// TwinCAT 3 PLC project RT1
// ProgramVersion: 3.1.4026.16
// libraries:
//   Tc2_Standard, * (Beckhoff Automation GmbH)
//   Tc2_System, * (Beckhoff Automation GmbH)
//   Tc2_Utilities, * (Beckhoff Automation GmbH)
//   Tc3_Module, * (Beckhoff Automation GmbH)
//   VisuDialogs, * (System)
// project tree:
//   DUTs/ ST_BasicStats.TcDUT
//   DUTs/Time/ E_WeekDay.TcDUT, stTimeToSchedule2.TcDUT, stTimeToSchedule3.TcDUT
//   / GlobalTextList.TcGTLO, PlcTask.TcTTO, Visualization Manager.TcVMO (not stored)
//   GVLs/ GVL_Const.TcGVL, GVL_TimeMeter.TcGVL, GVL_TimeSch.TcGVL
//   POUs/FBs/ FB_BasicStatistics.TcPOU, FB_HourMeter.TcPOU, FB_LastTimesStats.TcPOU, FB_TimeHandler.TcPOU, FB_BasicTimeScheduler.TcPOU, FB_UpdateTime.TcPOU
//   POUs/FUNs/ F_CmpTimeSchedule.TcPOU, F_CmpTimeStruct.TcPOU, F_DT_ToString.TcPOU
//   POUs/ MAIN.TcPOU, prgTimeHandler.TcPOU, prgTimeStatistics.TcPOU
//   VISUs/ EstatisticaTempo.TcVIS, FuncoesExtras.TcVIS, Hora.TcVIS, Data.TcVIS, ImagePool.TcIPO (not stored), Visualization.TcVIS, ProgramacaoHoraria.TcVIS
// real-time tasks:
//   TASK PlcTask: cycle T#10ms, priority 20, ADS port 351
//   TASK VISU_TASK: cycle T#200000us, priority 30, ADS port 350

CONFIGURATION RT1
    RESOURCE PLC ON TwinCAT3
        TASK PlcTask(INTERVAL := T#10ms, PRIORITY := 20);
        PROGRAM MAIN WITH PlcTask : MAIN;
    END_RESOURCE
END_CONFIGURATION

// ---- DUTs/ST_BasicStats.TcDUT
TYPE ST_BasicStats :
STRUCT
	minimum:LREAL;				//The mimimum of the distribution
	maximum:LREAL;              //The maximum of the distribution
	avg:LREAL;                  //The Average of the distribution
	variance:LREAL;             //The Variance
	standardDeviation:LREAL;    //Standard deviation
END_STRUCT
END_TYPE

// ---- DUTs/Time/E_WeekDay.TcDUT
TYPE E_WeekDay :
	(domingo:=0,
	segunda:=1,
	terca:=2,
	quarta:=3,
	quinta:=4,
	sexta:=5,
	sabado:=6);
END_TYPE

// ---- DUTs/Time/stTimeToSchedule2.TcDUT
TYPE stTimeToSchedule2 :
STRUCT
(*relacao do horario que a programacao horaria e ativa/desativada*)
	bIgnore:BOOL;		(*Relevante para desligar TRUE==>> nao desligar*)
	wHour:WORD;			(*Hora exata em que a saida sera acionada/desacionada*)
	wMinute:WORD;		(*Minuto exato em que a saida sera acionada/desacionada*)
	wSecond:WORD;		(*Segundo exato em que a saida sera acionada/desacionada*)
END_STRUCT
END_TYPE

// ---- DUTs/Time/stTimeToSchedule3.TcDUT
TYPE stTimeToSchedule3 :
STRUCT
	bUse:BOOL;			(*Relevante para desligar TRUE==>> nao desligar*)
	wHour:WORD;			(*Hora exata em que a saida sera acionada/desacionada*)
	wMinute:WORD;		(*Minuto exato em que a saida sera acionada/desacionada*)
	wSecond:WORD;		(*Segundo exato em que a saida sera acionada/desacionada*)	
END_STRUCT
END_TYPE

// ---- GVLs/GVL_Const.TcGVL
{attribute 'qualified_only'}
VAR_GLOBAL CONSTANT
	lastStatsValue:UDINT:=10;
END_VAR

// ---- GVLs/GVL_TimeMeter.TcGVL
{attribute 'qualified_only'}
VAR_GLOBAL
	enableTimeCount: BOOL;
	resetTimeCount: BOOL;
	currTaskTime:LREAL;
END_VAR
VAR_GLOBAL PERSISTENT
	hourCounting:LREAL;//
END_VAR

// ---- GVLs/GVL_TimeSch.TcGVL
{attribute 'qualified_only'}
VAR_GLOBAL CONSTANT
	cNumberOfEventSchedules:UINT:=8;//Quantidade de eventos necessarios/programados
(*Não alterar os valores daqui em diante*)
	ciSunday:WORD:=0;				//domingo
	ciMonday:WORD:=1;				//segunda
	ciTuesday:WORD:=2;				//terça
	ciWednesday:WORD:=3;			//quarta
	ciThursday:WORD:=4;				//quinta
	ciFriday:WORD:=5;				//sexta
	ciSaturday:WORD:=6;				//sabado
END_VAR
VAR_GLOBAL
	//Data e hora atuais
	actualDate:TIMESTRUCT;				//Data/Hora autais
	sActualDate: STRING;				(*String com a data atual*)
	sActualTime: STRING;				(*String com a hora atual*)
	sWeekDay:STRING;					(*Dia da semana*)
	//Acertar a hora
	timeToInsert: TIMESTRUCT;			//Hora a inserir (acertar hora)
	bUpdateTime: BOOL;					(*Atualizar a hora*)
	bUpdateDate: BOOL;					(*Atualizar a data*)
	(*Estrutura contendo a data e hora a serem inseridas*)	
	//Variaveis especificas da programacao horaria
	abOutScheduler:ARRAY[1..cNumberOfEventSchedules] OF BOOL;//Variaveis ativadas pelo bloco de programacao horaria
	uiIndexToCheck:UINT:=1;									//Index
	abErr:ARRAY[1..cNumberOfEventSchedules] OF BOOL;		//Erro na programacao horaria
	asErr:ARRAY[1..cNumberOfEventSchedules] OF STRING;		//
	bTurnOffOutput: BOOL;									//Desliga a saida dos blocos de 
END_VAR
VAR_GLOBAL PERSISTENT
	aTimeToSchActivate:ARRAY[0..6,1..cNumberOfEventSchedules] OF stTimeToSchedule3;		//Hora de ativar
	aTimeToSchDeactivate:ARRAY[0..6,1..cNumberOfEventSchedules] OF stTimeToSchedule3;	//Hora de desativar
END_VAR
//GVL_TimeSchBABR

// ---- POUs/MAIN.TcPOU
PROGRAM MAIN
VAR

END_VAR

prgTimeHandler();

prgTimeStatistics();

END_PROGRAM

// ---- POUs/prgTimeHandler.TcPOU
(*
	Programa realiza o gerenciamento da programacao horaria
	Esta rotina deve ser chamada no "MAIN" 
*)
PROGRAM prgTimeHandler
VAR
	timeScheduler:ARRAY[1..GVL_TimeSch.cNumberOfEventSchedules] OF FB_BasicTimeScheduler;
	i: UINT;
	timer:FB_TimeHandler;				(*Obtem a hora do sistema*)
	updateTime:FB_UpdateTime;			(*Bloco *)
	sActualTime: STRING;
	dt1: DATE_AND_TIME;
	timeMeter:FB_HourMeter;
	taskInfo: PlcTaskSystemInfo;
	bError: BOOL;
	sErr: STRING;
END_VAR

(*Le a data / Hora do sistema*)
timer(
	bDisplaySecond:= TRUE, 
	bShowDateNumberFormat:= TRUE, 
	sWeekDay=> GVL_TimeSch.sWeekDay, 
	sActualTime=> GVL_TimeSch.sActualTime, 
	sActualDate=> GVL_TimeSch.sActualDate, 
	outStruct=> GVL_TimeSch.actualDate);

(*Responsavel por atualizar a data/hora do sistema*)
updateTime(
	timeToInsert:= GVL_TimeSch.timeToInsert ,
	actualTime:= GVL_TimeSch.actualDate,
	bUpdateTime:= GVL_TimeSch.bUpdateTime,
	bUpdateDate:= GVL_TimeSch.bUpdateDate,
	bError=> ,
	iErrorId=> );

(*blocos de programacao horaria*)
FOR i := 1 TO GVL_TimeSch.cNumberOfEventSchedules DO
	timeScheduler[i](
		timeToActivate:= GVL_TimeSch.aTimeToSchActivate[GVL_TimeSch.actualDate.wDayOfWeek,i], 
		timeToDeactivate:= GVL_TimeSch.aTimeToSchDeactivate[GVL_TimeSch.actualDate.wDayOfWeek,i], 
		actualTime:= GVL_TimeSch.actualDate,
		bTurnOffOutput:= GVL_TimeSch.bTurnOffOutput,
		bErr=> GVL_TimeSch.abErr[i],
		sErr=> GVL_TimeSch.asErr[i],
		bOut=> GVL_TimeSch.abOutScheduler[i]);
END_FOR


taskInfo:=_TaskInfo[1];

sActualTime:=F_DT_ToString(dt1);

GVL_TimeMeter.currTaskTime:= UDINT_TO_LREAL(taskInfo.CycleTime)/10E6;

timeMeter(
	enableCount:= GVL_TimeMeter.enableTimeCount, 
	resetCount:= GVL_TimeMeter.resetTimeCount, 
	cycleTime:= GVL_TimeMeter.currTaskTime, 
	bError=>bError, 
	sErr=> sErr, 
	pastTime:=GVL_TimeMeter.hourCounting );

END_PROGRAM

// ---- POUs/FBs/FB_BasicTimeScheduler.TcPOU
FUNCTION_BLOCK FB_BasicTimeScheduler
VAR_INPUT
	timeToActivate:stTimeToSchedule3;		//Hora para ativar a saída
	timeToDeactivate:stTimeToSchedule3;		//Hora para desativar a saída
	actualTime:TIMESTRUCT;					//Hora/Data atual
	bTurnOffOutput:BOOL;					//Desliga a saída imediatamente
END_VAR
VAR_OUTPUT
	bErr: BOOL;
	sErr:STRING;
	bOut:BOOL;
END_VAR
VAR
	timeToActivateR_TRIG:R_TRIG;
	timeToDeactivateR_TRIG:R_TRIG;
END_VAR

sErr:='';
bErr:=FALSE;
IF NOT M_CheckTimeSchedule(timeToActivate) OR NOT (M_CheckTimeSchedule(timeToDeactivate) OR NOT timeToDeactivate.bUse) THEN
	bErr:=TRUE;
	sErr:='Parâmetros invalidos';
END_IF

timeToActivateR_TRIG(CLK:= M_CmpTimeStr_Schedule(actualTime,timeToActivate));
timeToDeactivateR_TRIG(CLK:= M_CmpTimeStr_Schedule(actualTime,timeToDeactivate));

IF timeToActivateR_TRIG.Q AND NOT bTurnOffOutput AND NOT bErr AND timeToActivate.bUse THEN
	bOut:=TRUE;
END_IF
IF timeToDeactivateR_TRIG.Q AND timeToDeactivate.bUse THEN
	bOut:=FALSE;
END_IF
IF bTurnOffOutput THEN
	bOut:=FALSE;
END_IF

METHOD M_CheckTimeSchedule : BOOL
VAR_INPUT
	timeSchedule:stTimeToSchedule3;	//Hora marcada a ser validada
END_VAR
M_CheckTimeSchedule:= (timeSchedule.wHour>=0 AND timeSchedule.wHour<=23)AND (timeSchedule.wMinute>=0 AND timeSchedule.wMinute <=59)
AND (timeSchedule.wSecond>=0 AND timeSchedule.wSecond <=59);
END_METHOD

METHOD PRIVATE M_CmpTimeStr_Schedule : BOOL
VAR_INPUT
	actualTime:TIMESTRUCT;
	scheduledTime:stTimeToSchedule3;
END_VAR
VAR
	timeToCmp:TIMESTRUCT;
END_VAR
(*
	Esse metodo retorna true caso a hora atual seja >= à hora marcada para ocorrer o evento
	Caso a variave 'bUse' do tempo marcado esteja desabilita também retorna false
*)
timeToCmp.wYear:=actualTime.wYear;
timeToCmp.wMonth:=actualTime.wMonth;
timeToCmp.wDay:=actualTime.wDay;
timeToCmp.wDayOfWeek:=actualTime.wDayOfWeek;
timeToCmp.wHour:=scheduledTime.wHour;
timeToCmp.wMinute:= scheduledTime.wMinute;
timeToCmp.wSecond:=scheduledTime.wSecond;
M_CmpTimeStr_Schedule:=F_CmpTimeStruct(actualTime,timeToCmp);
END_METHOD

END_FUNCTION_BLOCK

// ---- POUs/FUNs/F_CmpTimeStruct.TcPOU
FUNCTION F_CmpTimeStruct : BOOL
VAR_INPUT
	time1:TIMESTRUCT;
	time2:TIMESTRUCT;
END_VAR
VAR
END_VAR
(*Esta funcao verifica se a TimeStruct fornecida é válida
a variavel "time1"devera ser maior que a  variavel "time2" para que a funcao seja verdadeira*)

F_CmpTimeStruct:= SYSTEMTIME_TO_DT( time1)>SYSTEMTIME_TO_DT( time2);

END_FUNCTION

// ---- POUs/FBs/FB_TimeHandler.TcPOU
FUNCTION_BLOCK FB_TimeHandler
VAR_INPUT
	bDisplaySecond:BOOL;			(*Mostra os segundos na variavel de saida de hora*)
	bShowDateNumberFormat:BOOL;	(*Mostra a data em formato numerico (e.g.: 01/01/1970)*)
END_VAR
VAR_OUTPUT
	sActualMonth: STRING;			(*Mes do ano*)
	sWeekDay:STRING;				(*Dia da semana*)
	sActualTime:STRING;				(*Hora*)
	sActualDate:STRING;				(*Data atual*)
	outStruct:TIMESTRUCT;
END_VAR
VAR
	getTime:FB_LocalSystemTime;		(*Obtem a data/hora do sistema*)
	sSecond: STRING;
END_VAR


(*Obtem a hora do Windows*)
getTime(
	sNetID:='' ,
	bEnable:=TRUE ,
	dwCycle:= ,
	dwOpt:= ,
	tTimeout:= ,
	bValid=> ,
	tzID=> );

ASetStrings();
outStruct:=getTime.systemTime;

ACTION ASetStrings:
IF getTime.bValid THEN
	CASE getTime.systemTime.wMonth OF
		1:
			sActualMonth:='Janeiro';
		2:
			sActualMonth:='Fevereiro';
		3:
			sActualMonth:='Março';
		4:
			sActualMonth:='Abril';
		5:
			sActualMonth:='Maio';
		6:
			sActualMonth:='Junho';
		7:
			sActualMonth:='Julho';
		8:
			sActualMonth:='Agosto';
		9:
			sActualMonth:='Setembro';
		10:
			sActualMonth:='Outubro';
		11:
			sActualMonth:='Novembro';
		12:
			sActualMonth:='Dezembro';
	END_CASE

	CASE getTime.systemTime.wDayOfWeek OF
		0:
			sWeekDay:='Domingo';
		1:
			sWeekDay:='Segunda';
		2:
			sWeekDay:='Terça';
		3:
			sWeekDay:='Quarta';
		4:
			sWeekDay:='Quinta';
		5:
			sWeekDay:='Sexta';
		6:
			sWeekDay:='Sabado';
	END_CASE
	sSecond:=SEL(getTime.systemTime.wSecond<10,WORD_TO_STRING(getTime.systemTime.wSecond),CONCAT('0',WORD_TO_STRING(getTime.systemTime.wSecond)));

	sActualTime:=CONCAT(WORD_TO_STRING(getTime.systemTime.wHour),CONCAT(':',CONCAT(WORD_TO_STRING(getTime.systemTime.wMinute),SEL(bDisplaySecond,'',CONCAT(':',sSecond)))));

	IF NOT bShowDateNumberFormat THEN
		sActualDate:=CONCAT(WORD_TO_STRING(getTime.systemTime.wDay),CONCAT(' de ',CONCAT(sActualMonth,CONCAT(' de ' ,WORD_TO_STRING(getTime.systemTime.wYear)))));
	ELSE
		sActualDate:=CONCAT(WORD_TO_STRING(getTime.systemTime.wDay),CONCAT('/',CONCAT(WORD_TO_STRING(getTime.systemTime.wMonth),CONCAT('/',WORD_TO_STRING(getTime.systemTime.wYear)))));
	END_IF
ELSE
	sActualDate:='????';
	sActualTime:='????';
	sWeekDay:='????';
	sActualMonth:='????';
END_IF
END_ACTION

END_FUNCTION_BLOCK

// ---- POUs/FBs/FB_UpdateTime.TcPOU
FUNCTION_BLOCK FB_UpdateTime
VAR_INPUT
	timeToInsert:TIMESTRUCT;		(*estruta com data/hora a ser inserida*)
	actualTime:TIMESTRUCT;			(*estrutura contendo a data/hora atual*)
	bUpdateTime: BOOL;				(*atualiza a hora com um pulso nessa entrada*)
	bUpdateDate: BOOL;				(*atualiza a data com um pulso nessa entrada*)
END_VAR
VAR_OUTPUT
	bError: BOOL;						(*Erro ativo*)
	iErrorId: UDINT;					(*Id do erro*)
END_VAR
VAR
	setTime:NT_SetLocalTime;			(*Funcao para atualizar a data/hora*)
END_VAR

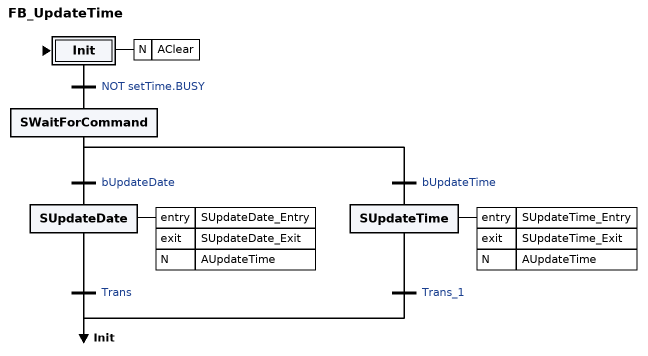
INITIAL_STEP Init:
    AClear(N);
END_STEP
TRANSITION FROM Init TO SWaitForCommand
    := NOT setTime.BUSY;
END_TRANSITION
STEP SWaitForCommand:
END_STEP
TRANSITION FROM SWaitForCommand TO SUpdateDate
    := bUpdateDate;
END_TRANSITION
STEP SUpdateDate:
    SUpdateDate_Entry(P1);  // entry action
    SUpdateDate_Exit(P0);  // exit action
    AUpdateTime(N);
END_STEP
TRANSITION FROM SUpdateDate TO Init
    := Trans;
END_TRANSITION
TRANSITION FROM SWaitForCommand TO SUpdateTime
    := bUpdateTime;
END_TRANSITION
STEP SUpdateTime:
    SUpdateTime_Entry(P1);  // entry action
    SUpdateTime_Exit(P0);  // exit action
    AUpdateTime(N);
END_STEP
TRANSITION FROM SUpdateTime TO Init
    := Trans_1;
END_TRANSITION

ACTION AClear:
setTime(	NETID:='' ,START:=FALSE );
END_ACTION

ACTION AUpdateTime:
setTime(
	NETID:='' ,
	START:= TRUE,
	ERR=>bError ,
	ERRID=> iErrorId);
END_ACTION

ACTION SUpdateDate_Entry:
(*Inicia o processo de atualizar a data*)


setTime.TIMESTR:=actualTime;
setTime.TIMESTR.wDay:=timeToInsert.wDay;
setTime.TIMESTR.wMonth:=timeToInsert.wMonth;
setTime.TIMESTR.wYear:=timeToInsert.wYear;
END_ACTION

ACTION SUpdateDate_Exit:
setTime(	NETID:='' ,START:=FALSE );
END_ACTION

ACTION SUpdateTime_Entry:
(*Inicia o processo de atualizar a data*)


setTime.TIMESTR:=actualTime;

setTime.TIMESTR.wHour:=timeToInsert.wHour;
setTime.TIMESTR.wMinute:=timeToInsert.wMinute;
setTime.TIMESTR.wSecond:=timeToInsert.wSecond;
END_ACTION

ACTION SUpdateTime_Exit:
setTime(	NETID:='' ,START:=FALSE );
END_ACTION

TRANSITION Trans:
NOT setTime.BUSY
END_TRANSITION

TRANSITION Trans_1:
NOT setTime.BUSY
END_TRANSITION

END_FUNCTION_BLOCK

// ---- POUs/FBs/FB_HourMeter.TcPOU
FUNCTION_BLOCK FB_HourMeter
VAR_INPUT
	enableCount: BOOL;	//this variable enables the time count
	resetCount:BOOL;	//set it to true in order to reset the whole count
	cycleTime:LREAL;	//cycle time in seconds
END_VAR
VAR_OUTPUT
	bError:BOOL;
	sErr:STRING;
END_VAR
VAR_IN_OUT
	pastTime:LREAL;	//Variable that contains the time past, should be persistent/retain outside the block otherwise the time count will not 
					//be kept once the PLC is stopped
END_VAR
VAR
	m:BOOL;			//memory to activate the rising trigger to reset the counter
END_VAR

IF enableCount AND cycleTime>0.0 THEN
	pastTime:= pastTime + cycleTime/3600;
	bError:=FALSE;
	sErr:='';
ELSIF cycleTime <=0 THEN
	bError:=TRUE;
	sErr:= 'wrong configured time';
END_IF


IF resetCount AND NOT m THEN
	pastTime:=0;
END_IF
m := resetCount;

END_FUNCTION_BLOCK

// ---- POUs/FUNs/F_DT_ToString.TcPOU
FUNCTION F_DT_ToString : STRING
VAR_INPUT
	in:DATE_AND_TIME;
END_VAR
VAR
	tsDtToConvert:TIMESTRUCT;
END_VAR

tsDtToConvert:= DT_TO_SYSTEMTIME(in);

F_DT_ToString:= CONCAT(WORD_TO_STRING(tsDtToConvert.wDay),'/');
F_DT_ToString:= CONCAT(F_DT_ToString, CONCAT( WORD_TO_STRING(tsDtToConvert.wMonth),'/'));
F_DT_ToString:= CONCAT(F_DT_ToString, CONCAT( WORD_TO_STRING(tsDtToConvert.wYear),'/'));
F_DT_ToString:= CONCAT(F_DT_ToString, ' ');
F_DT_ToString:= CONCAT(F_DT_ToString, CONCAT( WORD_TO_STRING(tsDtToConvert.wHour),':'));
F_DT_ToString:= CONCAT(F_DT_ToString, CONCAT( WORD_TO_STRING(tsDtToConvert.wMinute),':'));
F_DT_ToString:= CONCAT(F_DT_ToString,  WORD_TO_STRING(tsDtToConvert.wSecond));

END_FUNCTION

// ---- POUs/prgTimeStatistics.TcPOU
PROGRAM prgTimeStatistics
VAR
	enableTimeCount: BOOL;
	lastTimeStats:FB_LastTimesStats;
	stats:st_BasicStats;
	lastTime: TIME;
	currTime: TIME;
	lastTimes: ARRAY [1..GVL_Const.lastStatsValue] OF TIME;
	arLastTimes: ARRAY [1..GVL_Const.lastStatsValue] OF LREAL;
END_VAR

lastTimeStats(enable:= enableTimeCount,lastTime => lastTime, currTime=>currTime, lastTimes => lastTimes, arLastTimes => arLastTimes);

stats:=lastTimeStats.M_GetBasicStats();

END_PROGRAM

// ---- POUs/FBs/FB_LastTimesStats.TcPOU
FUNCTION_BLOCK FB_LastTimesStats EXTENDS FB_BasicStatistics
VAR_INPUT
	enable: BOOL;	//Enable time counting
END_VAR
VAR_OUTPUT
	lastTime:TIME;
	currTime:TIME;
	lastTimes:ARRAY[1..GVL_Const.lastStatsValue] OF TIME;
	arLastTimes:ARRAY[1..GVL_Const.lastStatsValue] OF LREAL;
END_VAR
VAR
	t1:TON;
	disableTrig:F_TRIG;
	i: UDINT;
END_VAR

disableTrig(CLK:= enable);
IF disableTrig.Q THEN
	lastTime:= t1.ET;
	FOR i:= GVL_Const.lastStatsValue TO 2 BY -1 DO
		lastTimes[i]:= lastTimes[i-1];
	END_FOR
	lastTimes[1]:=lastTime;
	FOR i:= 1 TO GVL_Const.lastStatsValue DO
		arLastTimes[i]:= TIME_TO_LREAL(lastTimes[i])/1000;
	END_FOR
END_IF
t1(IN:= enable, PT:= T#7D);
currTime:= t1.ET;

METHOD M_GetBasicStats : ST_BasicStats
VAR_INPUT
END_VAR
M_GetBasicStats.avg:=SUPER^.M_CalcAvg(THIS^.arLastTimes);
M_GetBasicStats.maximum:=SUPER^.M_CalcMax(THIS^.arLastTimes);
M_GetBasicStats.minimum:=SUPER^.M_CalcMin(THIS^.arLastTimes);
M_GetBasicStats.variance:=SUPER^.M_CalcVariance(THIS^.arLastTimes);
M_GetBasicStats.standardDeviation:=SUPER^.M_CalcSD(THIS^.arLastTimes);
END_METHOD

END_FUNCTION_BLOCK

// ---- POUs/FBs/FB_BasicStatistics.TcPOU
FUNCTION_BLOCK FB_BasicStatistics
VAR_INPUT
END_VAR
VAR_OUTPUT
END_VAR
VAR
END_VAR

METHOD M_CalcAvg : LREAL
VAR_IN_OUT
	valuesToAvg:ARRAY[*] OF LREAL;
END_VAR
VAR
	i: DINT;
	sum:LREAL;
	numOfElements: LREAL;
END_VAR
sum:=0;
numOfElements:=0;
FOR i := LOWER_BOUND(valuesToAvg,1) TO UPPER_BOUND(valuesToAvg,1) DO
	sum:= sum+ valuesToAvg[i];
	numOfElements:=numOfElements+1;
END_FOR
IF numOfElements >0 THEN
	M_CalcAvg :=sum/numOfElements;
END_IF
END_METHOD

METHOD M_CalcMax : LREAL
VAR_IN_OUT
	valuesToMax:ARRAY[*] OF LREAL;
END_VAR

VAR
	maximum: LREAL;
	i: DINT;
END_VAR
maximum:=valuesToMax[1];
FOR i:= LOWER_BOUND(valuesToMax,1) TO UPPER_BOUND(valuesToMax,1) DO
	maximum:= MAX(maximum,valuesToMax[i]);
END_FOR
M_CalcMax:= maximum;
END_METHOD

METHOD M_CalcMin : LREAL
VAR_IN_OUT
	valuesToMin:ARRAY[*] OF LREAL;
END_VAR

VAR
	minimum: LREAL;
	i: DINT;
END_VAR
minimum:=valuesToMin[1];
FOR i:= LOWER_BOUND(valuesToMin,1) TO UPPER_BOUND(valuesToMin,1) DO
	minimum:= MIN(minimum,valuesToMin[i]);
END_FOR
M_CalcMin:= minimum;
END_METHOD

METHOD M_CalcSD : LREAL
VAR_INPUT
	valuesToSD:ARRAY[1..GVL_Const.lastStatsValue] OF LREAL;
END_VAR
M_CalcSD := SQRT(M_CalcVariance(valuesToSD));
END_METHOD

METHOD PUBLIC M_CalcVariance : LREAL
VAR_IN_OUT
	valuesToVar:ARRAY[*] OF LREAL;
END_VAR
VAR
	i: DINT;
	sum:LREAL;
	avg:LREAL;
	numOfElements:lreal;
END_VAR
sum:=numOfElements:=0;
avg:= M_CalcAvg(valuesToVar);
FOR i := LOWER_BOUND(valuesToVar,1) TO UPPER_BOUND(valuesToVar,1) DO
	sum:= sum+EXPT(valuesToVar[i]-avg,2);
	numOfElements:= numOfElements+1;
END_FOR
M_CalcVariance:= sum/numOfElements;
END_METHOD

END_FUNCTION_BLOCK

// ---- POUs/FUNs/F_CmpTimeSchedule.TcPOU
FUNCTION F_CmpTimeSchedule : BOOL
VAR_INPUT
	timeToActivate:stTimeToSchedule2;	(*Hora para ligar a saida*)
	timeToDeactivate:stTimeToSchedule2;	(*Hora para desligar a saida*)
END_VAR
VAR
END_VAR

F_CmpTimeSchedule:=(timeToDeactivate.wHour>timeToActivate.wHour) OR ((timeToDeactivate.wHour = timeToActivate.wHour) AND (timeToDeactivate.wMinute> timeToActivate.wMinute));

END_FUNCTION

// ---- GlobalTextList.TcGTLO
TEXTLIST GlobalTextList
  148 = '%.1f'
  509 = '%d'
  18 = '%s'
  793 = '%t'
  615 = '180'
  9 = 'Acertar Data'
  8 = 'Acertar Hora'
  12 = 'Ano'
  19 = 'Ativar'
  88 = 'Atual'
  7 = 'Atualizar'
  16 = 'Checkbox'
  0 = 'DATA : %s'
  20 = 'Desativar'
  183 = 'Desvio P.'
  14 = 'dia'
  15 = 'Dia'
  28 = 'Dia : %s'
  26 = 'domingo'
  27 = 'Domingo'
  585 = 'Estats tempo'
  694 = 'Extras'
  986 = 'Habilitar'
  4 = 'Hora'
  1 = 'HORA : %s'
  891 = 'Horas : %.1f'
  13 = 'Mes'
  5 = 'Min'
  876 = 'Máximo'
  277 = 'Médio'
  38 = 'Mínimo'
  783 = 'Programação'
  252 = 'Programação horária'
  22 = 'Quarta'
  23 = 'Quinta'
  287 = 'Reset'
  25 = 'Sabado'
  6 = 'Seg'
  17 = 'Segunda'
  24 = 'Sexta'
  610 = 'T. Ciclo %.2f (s)'
  11 = 'Tela 1'
  10 = 'Tela 2'
  21 = 'Terça'
  3 = 'Update Date'
  2 = 'Update Time'
  181 = 'Variância'
  250 = 'Último'
  665 = 'Últimos tempos'
  29 = 'Últimos tempos (Real)'
  583 = 'Últimos tempos (s)'
  391 = 'Últimos tempos (Segundos)'
  880 = 'Últimos tempos (T)'
END_TEXTLIST

// ---- VISUs/EstatisticaTempo.TcVIS
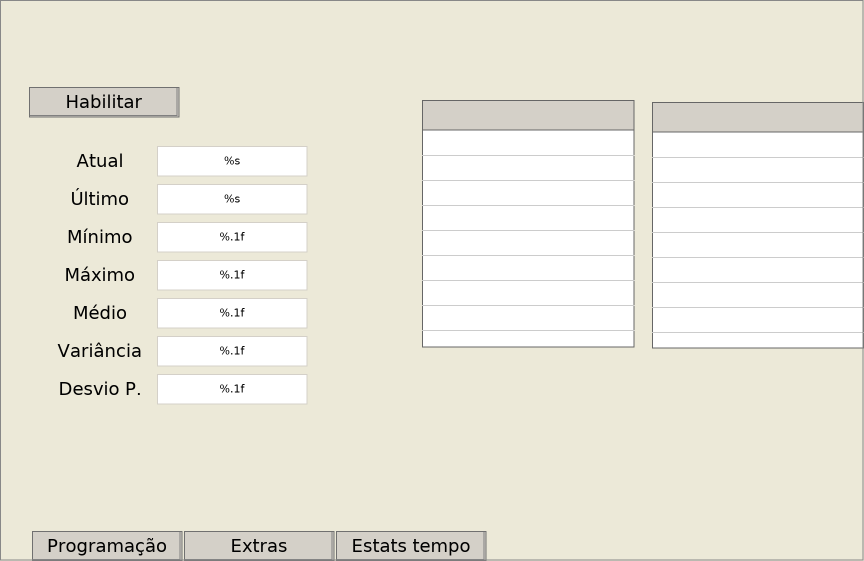
VISUALIZATION EstatisticaTempo  // 864x561
    Button (32,531 150x30), "Programação"
        OnMouseClick: change screen: Visualization
    Button (184,531 150x30), "Extras"
        OnMouseClick: change screen: FuncoesExtras
    Button (336,531 150x30), "Estats tempo"
        OnMouseClick: change screen: EstatisticaTempo
    Table (422,100 212x247), data array: prgTimeStatistics.lastTimes
        p3854506369: prgTimeStatistics.lastTimes[INDEX]
        p2232123230: Últimos tempos (T)
    Table (652,102 212x246), data array: prgTimeStatistics.arLastTimes
        p3854506369: prgTimeStatistics.arLastTimes[INDEX]
        p2232123230: Últimos tempos (s)
    Button (29,87 150x30), "Habilitar"
        toggle prgTimeStatistics.enableTimeCount
    Label (40,146 120x30), "Atual"
    Label (40,184 120x30), "Último"
    Label (40,222 120x30), "Mínimo"
    Label (40,260 120x30), "Máximo"
    Label (40,298 120x30), "Médio"
    Label (40,336 120x30), "Variância"
    Label (40,374 120x30), "Desvio P."
    Textfield (157,146 150x30), "%s", text variable: prgTimeStatistics.lastTimeStats.currTime
    Textfield (157,184 150x30), "%s", text variable: prgTimeStatistics.lastTimeStats.lastTime
    Textfield (157,222 150x30), "%.1f", text variable: prgTimeStatistics.stats.minimum
    Textfield (157,260 150x30), "%.1f", text variable: prgTimeStatistics.stats.maximum
    Textfield (157,298 150x30), "%.1f", text variable: prgTimeStatistics.stats.avg
    Textfield (157,336 150x30), "%.1f", text variable: prgTimeStatistics.stats.variance
    Textfield (157,374 150x30), "%.1f", text variable: prgTimeStatistics.stats.standardDeviation
END_VISUALIZATION

// ---- VISUs/FuncoesExtras.TcVIS
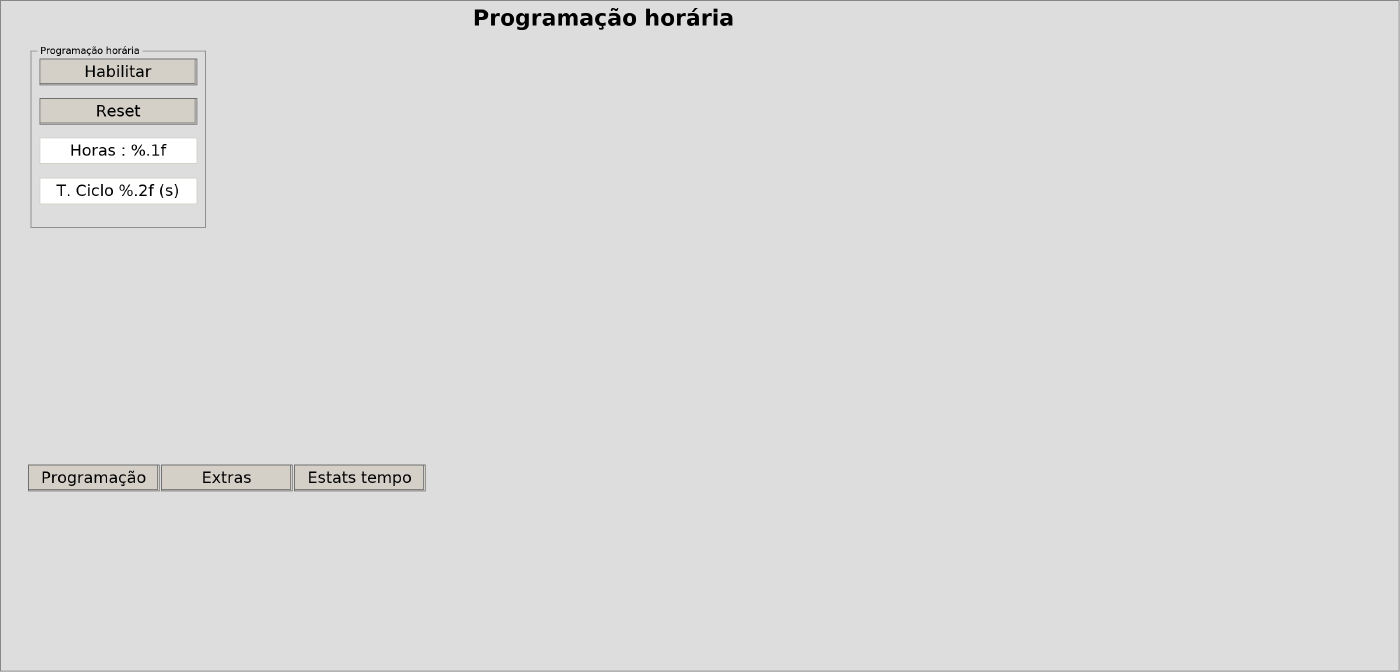
VISUALIZATION FuncoesExtras  // 1600x768
    Label (500,5 380x30), "Programação horária"
    GroupBox (35,50 200x210), "Programação horária"
        Button (10,17 180x30), "Habilitar"
            toggle GVL_TimeMeter.enableTimeCount
        Button (10,62 180x30), "Reset"
            tap GVL_TimeMeter.resetTimeCount
        Textfield (10,107 180x30), "Horas : %.1f", text variable: GVL_TimeMeter.hourCounting
        Textfield (10,153 180x30), "T. Ciclo %.2f (s)", text variable: GVL_TimeMeter.currTaskTime
    Button (32,531 150x30), "Programação"
        OnMouseClick: change screen: Visualization
    Button (184,531 150x30), "Extras"
        OnMouseClick: change screen: FuncoesExtras
    Button (336,531 150x30), "Estats tempo"
        OnMouseClick: change screen: EstatisticaTempo
END_VISUALIZATION

// ---- VISUs/Hora.TcVIS
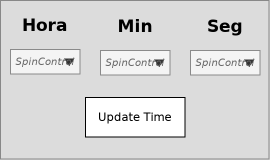
VISUALIZATION Hora  // 270x160
    Rectangle (85,97 100x40), "Update Time"
        tap GVL_TimeSch.bUpdateTime
    SpinControl (10,49 70x25), variable: GVL_TimeSch.timeToInsert.wHour
        OnMouseClick: write the text variable via Default, min 0, max 23
    Label (10,10 70x30), "Hora"
    SpinControl (100,50 70x25), variable: GVL_TimeSch.timeToInsert.wMinute
        OnMouseClick: write the text variable via Default, min 0, max 59
    Label (100,11 70x30), "Min"
    SpinControl (190,50 70x25), variable: GVL_TimeSch.timeToInsert.wSecond
        OnMouseClick: write the text variable via Default, min 0, max 59
    Label (190,11 70x30), "Seg"
END_VISUALIZATION

// ---- VISUs/Data.TcVIS
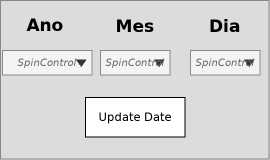
VISUALIZATION Data  // 270x160
    SpinControl (2,50 90x25), variable: GVL_TimeSch.timeToInsert.wYear
        OnMouseClick: write the text variable via Default, min 2000, max 3000
    Label (10,10 70x30), "Ano"
    SpinControl (100,50 70x25), variable: GVL_TimeSch.timeToInsert.wMonth
        OnMouseClick: write the text variable via Default, min 1, max 12
    Label (100,11 70x30), "Mes"
    SpinControl (190,50 70x25), variable: GVL_TimeSch.timeToInsert.wDay
        OnMouseClick: write the text variable via Default, min 1, max 31
    Label (190,11 70x30), "Dia"
    Rectangle (85,97 100x40), "Update Date"
        tap GVL_TimeSch.bUpdateDate
END_VISUALIZATION

// ---- VISUs/Visualization.TcVIS
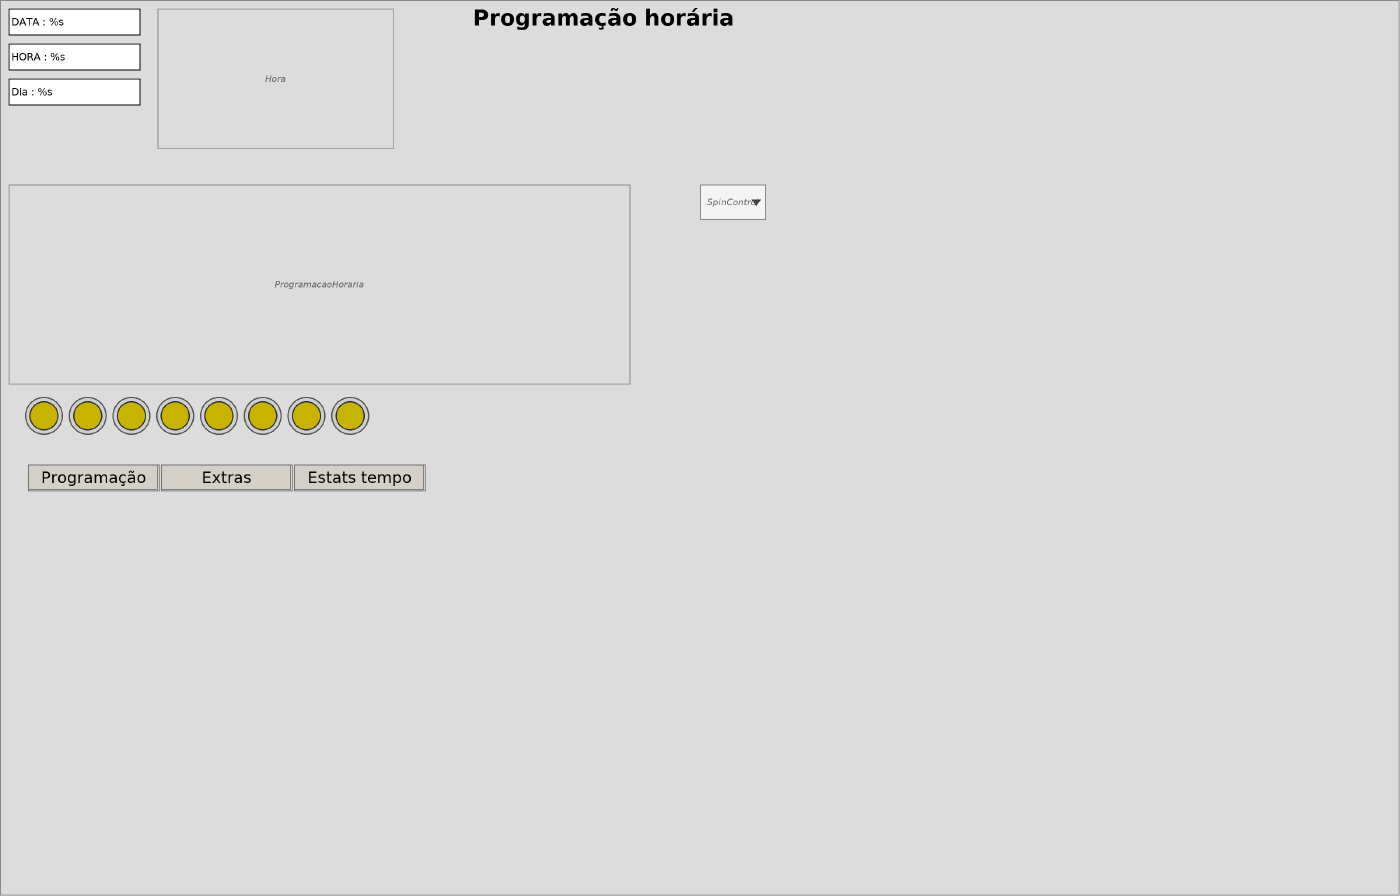
VISUALIZATION Visualization  // 1600x1024
    Rectangle (10,10 150x30), "DATA : %s", text variable: GVL_TimeSch.sActualDate
    Rectangle (10,50 150x30), "HORA : %s", text variable: GVL_TimeSch.sActualTime
    TabControl (180,10 270x160)
        shows Hora()
        shows Data()
        [0]: TabTitle=Acertar Hora
        [1]: TabTitle=Acertar Data
    TabControl (10,211 710x228)
        shows ProgramacaoHoraria(uiIndex := GVL_TimeSch.uiIndexToCheck, wDayOfWeek := GVL_TimeSch.ciMonday)
        shows ProgramacaoHoraria(uiIndex := GVL_TimeSch.uiIndexToCheck, wDayOfWeek := GVL_TimeSch.ciTuesday)
        shows ProgramacaoHoraria(uiIndex := GVL_TimeSch.uiIndexToCheck, wDayOfWeek := GVL_TimeSch.ciWednesday)
        shows ProgramacaoHoraria(uiIndex := GVL_TimeSch.uiIndexToCheck, wDayOfWeek := GVL_TimeSch.ciThursday)
        shows ProgramacaoHoraria(uiIndex := GVL_TimeSch.uiIndexToCheck, wDayOfWeek := GVL_TimeSch.ciFriday)
        shows ProgramacaoHoraria(uiIndex := GVL_TimeSch.uiIndexToCheck, wDayOfWeek := GVL_TimeSch.ciSaturday)
        shows ProgramacaoHoraria(uiIndex := GVL_TimeSch.uiIndexToCheck, wDayOfWeek := GVL_TimeSch.ciSunday)
        [0]: TabTitle=Segunda
        [1]: TabTitle=Terça
        [2]: TabTitle=Quarta
        [3]: TabTitle=Quinta
        [4]: TabTitle=Sexta
        [5]: TabTitle=Sabado
        [6]: TabTitle=Domingo
    Rectangle (10,90 150x30), "Dia : %s", text variable: GVL_TimeSch.sWeekDay
    SpinControl (800,211 75x40), variable: GVL_TimeSch.uiIndexToCheck
        p651134158: GVL_TimeSch.cNumberOfEventSchedules
    Group (25,450 400x50)
        Lamp1 (0,0 50x50), variable: GVL_TimeSch.abOutScheduler[1], style: Lamp-Lamp1-Yellow
        Lamp1 (50,0 50x50), variable: GVL_TimeSch.abOutScheduler[2], style: Lamp-Lamp1-Yellow
        Lamp1 (100,0 50x50), variable: GVL_TimeSch.abOutScheduler[3], style: Lamp-Lamp1-Yellow
        Lamp1 (150,0 50x50), variable: GVL_TimeSch.abOutScheduler[4], style: Lamp-Lamp1-Yellow
        Lamp1 (200,0 50x50), variable: GVL_TimeSch.abOutScheduler[5], style: Lamp-Lamp1-Yellow
        Lamp1 (250,0 50x50), variable: GVL_TimeSch.abOutScheduler[6], style: Lamp-Lamp1-Yellow
        Lamp1 (300,0 50x50), variable: GVL_TimeSch.abOutScheduler[7], style: Lamp-Lamp1-Yellow
        Lamp1 (350,0 50x50), variable: GVL_TimeSch.abOutScheduler[8], style: Lamp-Lamp1-Yellow
    Label (500,5 380x30), "Programação horária"
    Button (32,531 150x30), "Programação"
        OnMouseClick: change screen: Visualization
    Button (184,531 150x30), "Extras"
        OnMouseClick: change screen: FuncoesExtras
    Button (336,531 150x30), "Estats tempo"
        OnMouseClick: change screen: EstatisticaTempo
END_VISUALIZATION

// ---- VISUs/ProgramacaoHoraria.TcVIS
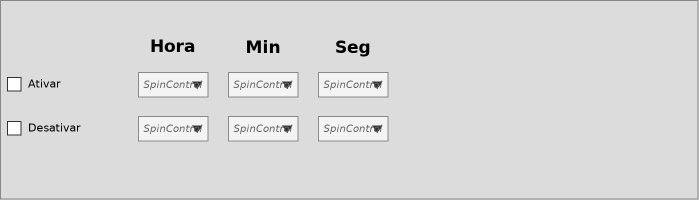
VISUALIZATION ProgramacaoHoraria  // 699x200
VAR_IN_OUT

END_VAR
VAR_INPUT
	uiIndex:UINT;		//Indice da programacao horaria
	wDayOfWeek:WORD;	
END_VAR
    Checkbox (5,69 120x30), "Ativar", variable: GVL_TimeSch.aTimeToSchActivate[wDayOfWeek,uiIndex].bUse
    Checkbox (5,113 120x30), "Desativar", variable: GVL_TimeSch.aTimeToSchDeactivate[wDayOfWeek,uiIndex].bUse
    SpinControl (138,72 70x25), variable: GVL_TimeSch.aTimeToSchActivate[wDayOfWeek,uiIndex].wHour
        OnMouseClick: write the text variable via Default, min 0, max 23
    Label (138,31 70x30), "Hora"
    SpinControl (228,72 70x25), variable: GVL_TimeSch.aTimeToSchActivate[wDayOfWeek,uiIndex].wMinute
        OnMouseClick: write the text variable via Default, min 0, max 59
    Label (228,32 70x30), "Min"
    SpinControl (318,72 70x25), variable: GVL_TimeSch.aTimeToSchActivate[wDayOfWeek,uiIndex].wSecond
        OnMouseClick: write the text variable via Default, min 0, max 59
    Label (318,32 70x30), "Seg"
    SpinControl (138,116 70x25), variable: GVL_TimeSch.aTimeToSchDeactivate[wDayOfWeek,uiIndex].wHour
        OnMouseClick: write the text variable via Default, min 0, max 23
    SpinControl (228,116 70x25), variable: GVL_TimeSch.aTimeToSchDeactivate[wDayOfWeek,uiIndex].wMinute
        OnMouseClick: write the text variable via Default, min 0, max 59
    SpinControl (318,116 70x25), variable: GVL_TimeSch.aTimeToSchDeactivate[wDayOfWeek,uiIndex].wSecond
        OnMouseClick: write the text variable via Default, min 0, max 59
END_VISUALIZATION
